{attribute addProperty BoxType "ELX9560-0000-0018"}
{attribute addProperty Id "Status_UinAT %I*Status_Uin_51406150810Status_UexAT %I*Status_Uex_A3DD649E810WcStateAT %I*WcState_98A4DF7520.250InfoDataAT %I*InfoData_192954DE1620"}
{attribute addProperty CRC "1879269500"}
{attribute addProperty SizeInBites "34"}
{attribute addProperty SizeInBytes "4.25"}
TYPE ELX9560_AB2C9EC5 :
STRUCT
	{attribute addProperty Name "Status_Uin"}
	Status_Uin : Status_Uin_51406150;
	{attribute addProperty Name "Status_Uex"}
	Status_Uex : Status_Uex_A3DD649E;
	{attribute addProperty Name "WcState"}
	WcState : WcState_98A4DF75;
	{attribute addProperty Name "InfoData"}
	InfoData : InfoData_192954DE;
END_STRUCT
END_TYPE

(* stored: Version 1.2.0.0, ProductVersion 3.1.4024.9
   DUT ELX9560_AB2C9EC5: Id {b4050158-4f7d-45f8-aacd-08f5f8acd258} *)
